// TIA Portal V17 export
// export: Created 2023-05-07T12:12:22.5026465Z, ExportSetting WithDefaults, DisplayName Totally Integrated Automation Portal, DisplayVersion V17, DisplayName TIA Portal Openness, DisplayVersion V17, DisplayName TIA Portal Version Control Interface, DisplayVersion V17, DisplayName TIA Portal Test Suite Advanced, DisplayVersion V17, DisplayName STEP 7 Professional, DisplayVersion V17, DisplayName SIMATIC Energy Suite, DisplayVersion V17, DisplayName STEP 7 Safety, DisplayVersion V17, DisplayName WinCC Professional, DisplayVersion V17
DATA_BLOCK "RegSugeno_DB"   // DB7
VERSION : 0.1
// stored: AutoNumber true, InstanceOfName Takagi-SugenoFuzzy-PI, InstanceOfType FB
"Takagi-SugenoFuzzy-PI"
   // VAR_INPUT
   //    PV : Real;
   //    SP : Real;
   // END_VAR
   // VAR_OUTPUT
   //    MV : Real;
   // END_VAR
   // VAR
   //    n_e : Real;
   //    i_e : Real;
   //    ni_e : Real;
   // END_VAR
BEGIN
END_DATA_BLOCK
